// TIA Portal V17 export
// export: Created 2023-12-22T15:08:09.8498698Z, ExportSetting WithDefaults, DisplayName Totally Integrated Automation Portal, DisplayVersion V17, DisplayName TIA Portal Openness, DisplayVersion V17, DisplayName TIA Portal Version Control Interface, DisplayVersion V17, DisplayName STEP 7 Professional, DisplayVersion V17, DisplayName STEP 7 Safety, DisplayVersion V17, DisplayName WinCC Advanced, DisplayVersion V17
DATA_BLOCK "LE_Diag_DB"   // DB5
VERSION : 0.1
// stored: AutoNumber true, DBAccessibleFromOPCUA true, DBAccessibleFromWebserver true, InstanceOfName LE_Diag, InstanceOfType FB
"LE_Diag"
   // VAR_OUTPUT
   //    LE : Real;
   // END_VAR
   // VAR
   //    Select : Int;
   // END_VAR
   // VAR RETAIN
   //    Use { S7_SetPoint := 'True'} : Array[0..5] of Bool;
   // END_VAR
   // VAR
   //    LEx : Array[0..5] of Real;
   //    Delta : Array[0..5] of Real;
   // END_VAR
   // VAR RETAIN
   //    Delta_Max { S7_SetPoint := 'True'} : Real := 0.1;
   // END_VAR
   // VAR
   //    Warning : Array[0..15] of Bool;
   //    cnt : Int;
   //    w_word : Int;
   // END_VAR
BEGIN
   Use[0] := FALSE;
   Use[1] := TRUE;
   Use[2..5] := FALSE;
END_DATA_BLOCK
